FUNCTION F_CheckStepperAlarmsAcked : BOOL
VAR_INPUT
    nRail : SINT;              // Rail number (1, 2, 3, or 4)
END_VAR
VAR
    bAllAlarmsAcked : BOOL := TRUE;
END_VAR

// ============================================================================
// VALIDATE RAIL NUMBER
// ============================================================================
IF nRail < 1 OR nRail > 4 THEN
    F_CheckStepperAlarmsAcked := FALSE;
    RETURN;
END_IF

// ============================================================================
// CHECK ALL STEPPER ALARMS FOR THIS RAIL ARE ACKNOWLEDGED
// ============================================================================
CASE nRail OF
    1: // Rail 1 stepper alarms
        bAllAlarmsAcked := bAllAlarmsAcked AND GVL_Alarms.R1_Stepper_Motion_Failed.bAcked;
        bAllAlarmsAcked := bAllAlarmsAcked AND GVL_Alarms.R1_Stepper_Homing_Failed.bAcked;
        bAllAlarmsAcked := bAllAlarmsAcked AND GVL_Alarms.R1_Stepper_Homing_Interrupted.bAcked;
        bAllAlarmsAcked := bAllAlarmsAcked AND GVL_Alarms.R1_Stepper_Motion_Interrupted.bAcked;
        bAllAlarmsAcked := bAllAlarmsAcked AND GVL_Alarms.R1_Stepper_PowerUp_Failed.bAcked;
        bAllAlarmsAcked := bAllAlarmsAcked AND GVL_Alarms.R1_Stepper_Reset_Failed.bAcked;
        
    2: // Rail 2 stepper alarms
        bAllAlarmsAcked := bAllAlarmsAcked AND GVL_Alarms.R2_Stepper_PowerUp_Failed.bAcked;
        bAllAlarmsAcked := bAllAlarmsAcked AND GVL_Alarms.R2_Stepper_Homing_Failed.bAcked;
        bAllAlarmsAcked := bAllAlarmsAcked AND GVL_Alarms.R2_Stepper_Homing_Interrupted.bAcked;
        bAllAlarmsAcked := bAllAlarmsAcked AND GVL_Alarms.R2_Stepper_Motion_Failed.bAcked;
        bAllAlarmsAcked := bAllAlarmsAcked AND GVL_Alarms.R2_Stepper_Motion_Interrupted.bAcked;
        bAllAlarmsAcked := bAllAlarmsAcked AND GVL_Alarms.R2_Stepper_Reset_Failed.bAcked;
        
    3: // Rail 3 stepper alarms
        bAllAlarmsAcked := bAllAlarmsAcked AND GVL_Alarms.R3_Stepper_PowerUp_Failed.bAcked;
        bAllAlarmsAcked := bAllAlarmsAcked AND GVL_Alarms.R3_Stepper_Homing_Failed.bAcked;
        bAllAlarmsAcked := bAllAlarmsAcked AND GVL_Alarms.R3_Stepper_Homing_Interrupted.bAcked;
        bAllAlarmsAcked := bAllAlarmsAcked AND GVL_Alarms.R3_Stepper_Motion_Failed.bAcked;
        bAllAlarmsAcked := bAllAlarmsAcked AND GVL_Alarms.R3_Stepper_Motion_Interrupted.bAcked;
        bAllAlarmsAcked := bAllAlarmsAcked AND GVL_Alarms.R3_Stepper_Reset_Failed.bAcked;
        
    4: // Rail 4 stepper alarms
        bAllAlarmsAcked := bAllAlarmsAcked AND GVL_Alarms.R4_Stepper_PowerUp_Failed.bAcked;
        bAllAlarmsAcked := bAllAlarmsAcked AND GVL_Alarms.R4_Stepper_Homing_Failed.bAcked;
        bAllAlarmsAcked := bAllAlarmsAcked AND GVL_Alarms.R4_Stepper_Homing_Interrupted.bAcked;
        bAllAlarmsAcked := bAllAlarmsAcked AND GVL_Alarms.R4_Stepper_Motion_Failed.bAcked;
        bAllAlarmsAcked := bAllAlarmsAcked AND GVL_Alarms.R4_Stepper_Motion_Interrupted.bAcked;
        bAllAlarmsAcked := bAllAlarmsAcked AND GVL_Alarms.R4_Stepper_Reset_Failed.bAcked;
        
    ELSE
        bAllAlarmsAcked := FALSE; // Invalid rail number
END_CASE

F_CheckStepperAlarmsAcked := bAllAlarmsAcked;

END_FUNCTION

(* stored: Version 1.1.0.1, ProductVersion 3.1.4026.11
   POU F_CheckStepperAlarmsAcked: Id {baa63939-bcb8-4184-bbb9-984588a51a1b}, SpecialFunc None *)
